# EPICS substitutions: dh2000Sup/error_setter.substitutions
# Errors are not forwarded in protocol redirects

file $(UTILITIES)/db/error_setter.template {
  pattern
    {P, STREAM_PV, PV_NAME}

    {"\$(P)", "SHUTTER:STATUS", "INTERLOCK"}
}
